(* IEC 61131-3 sources: SafePLC-Gen-Evaluation/Evaluation Results/P_ID/run_01, 2 files *)

(* ---- io_declarations.st ---- *)
(* ==================================================  *)
(* PLC I/O Variable Declarations — CODESYS 3.5  *)
(* Generated by SafePLC-Gen Multimodal  *)
(* ==================================================  *)

VAR_GLOBAL
    (* --- Analog Inputs ---  *)
    FT_10_Raw                    AT %IW0       : INT := 0;    (* FT-10 — Flow transmitter on upper feed line, mea  *)
    FT_11_Raw                    AT %IW2       : INT := 0;    (* FT-11 — Flow transmitter on lower feed line, mea  *)
    (* --- Analog Outputs ---  *)
    Fv_3_3040_Out                AT %QW0       : INT := 0;    (* Fv-3-3040 — Flow control valve on upper feed line fr  *)
    Fv_3_3041_Out                AT %QW2       : INT := 0;    (* Fv-3-3041 — Flow control valve on lower feed line fr  *)
END_VAR

(* ---- generated_code.st ---- *)
(* Generated by SafePLC-Gen Multimodal — CODESYS 3.5 *)
(* IEC 61131-3 Structured Text *)
(* Date: 2026-04-25T12:45:35.863016 *)

PROGRAM FlowControl

VAR
    FT_10_Raw                    AT %IW0       : INT := 0;
    FT_11_Raw                    AT %IW2       : INT := 0;
    Fv_3_3040_Out                AT %QW0       : INT := 0;
    Fv_3_3041_Out                AT %QW2       : INT := 0;
END_VAR

VAR
    FT_10_Scaled                 : REAL := 0.0;
    FT_11_Scaled                 : REAL := 0.0;

    FT_10_HH_SP                  : REAL := 180.0;
    FT_10_H_SP                   : REAL := 160.0;
    FT_10_L_SP                   : REAL := 40.0;
    FT_10_LL_SP                  : REAL := 20.0;
    FT_10_Deadband               : REAL := 5.0;
    FT_10_H                      : BOOL := FALSE;
    FT_10_L                      : BOOL := FALSE;
    FT_10_HH_Latch               : SR := (S1 := FALSE, R := FALSE, Q1 := FALSE);
    FT_10_LL_Latch               : SR := (S1 := FALSE, R := FALSE, Q1 := FALSE);
    FT_10_HH_Ack                 : BOOL := FALSE;
    FT_10_LL_Ack                 : BOOL := FALSE;

    FT_11_HH_SP                  : REAL := 180.0;
    FT_11_H_SP                   : REAL := 160.0;
    FT_11_L_SP                   : REAL := 40.0;
    FT_11_LL_SP                  : REAL := 20.0;
    FT_11_Deadband               : REAL := 5.0;
    FT_11_H                      : BOOL := FALSE;
    FT_11_L                      : BOOL := FALSE;
    FT_11_HH_Latch               : SR := (S1 := FALSE, R := FALSE, Q1 := FALSE);
    FT_11_LL_Latch               : SR := (S1 := FALSE, R := FALSE, Q1 := FALSE);
    FT_11_HH_Ack                 : BOOL := FALSE;
    FT_11_LL_Ack                 : BOOL := FALSE;

    FT_10_SP                     : REAL := 100.0;
    FT_10_Kp                     : REAL := 1.2;
    FT_10_Ki                     : REAL := 0.05;
    FT_10_Error                  : REAL := 0.0;
    FT_10_Integral               : REAL := 0.0;
    FT_10_Output                 : REAL := 0.0;

    FT_11_SP                     : REAL := 100.0;
    FT_11_Kp                     : REAL := 1.2;
    FT_11_Ki                     : REAL := 0.05;
    FT_11_Error                  : REAL := 0.0;
    FT_11_Integral               : REAL := 0.0;
    FT_11_Output                 : REAL := 0.0;

    System_Alarm                 : BOOL := FALSE;
    FirstScan                    : BOOL := TRUE;
END_VAR

IF FirstScan THEN
    Fv_3_3040_Out  := 6554;
    Fv_3_3041_Out  := 6554;
    FT_10_Integral := 0.0;
    FT_11_Integral := 0.0;
    FirstScan      := FALSE;
    RETURN;
END_IF;

FT_10_Scaled := ((INT_TO_REAL(FT_10_Raw) - 6554.0) / (32767.0 - 6554.0)) * 200.0;
FT_11_Scaled := ((INT_TO_REAL(FT_11_Raw) - 6554.0) / (32767.0 - 6554.0)) * 200.0;

(* FT-10 HH latch *)
IF FT_10_Scaled >= FT_10_HH_SP THEN
    FT_10_HH_Latch.S1 := TRUE;
ELSIF FT_10_Scaled <= (FT_10_HH_SP - FT_10_Deadband) THEN
    FT_10_HH_Latch.S1 := FALSE;
END_IF;
FT_10_HH_Latch.R := FT_10_HH_Ack AND (FT_10_Scaled < FT_10_HH_SP);
FT_10_HH_Latch(S1 := FT_10_HH_Latch.S1, R := FT_10_HH_Latch.R);

(* FT-10 H alarm *)
IF FT_10_Scaled >= FT_10_H_SP THEN
    FT_10_H := TRUE;
ELSIF FT_10_Scaled <= (FT_10_H_SP - FT_10_Deadband) THEN
    FT_10_H := FALSE;
END_IF;

(* FT-10 L alarm *)
IF FT_10_Scaled <= FT_10_L_SP THEN
    FT_10_L := TRUE;
ELSIF FT_10_Scaled >= (FT_10_L_SP + FT_10_Deadband) THEN
    FT_10_L := FALSE;
END_IF;

(* FT-10 LL latch *)
IF FT_10_Scaled <= FT_10_LL_SP THEN
    FT_10_LL_Latch.S1 := TRUE;
ELSIF FT_10_Scaled >= (FT_10_LL_SP + FT_10_Deadband) THEN
    FT_10_LL_Latch.S1 := FALSE;
END_IF;
FT_10_LL_Latch.R := FT_10_LL_Ack AND (FT_10_Scaled > FT_10_LL_SP);
FT_10_LL_Latch(S1 := FT_10_LL_Latch.S1, R := FT_10_LL_Latch.R);

(* FT-11 HH latch *)
IF FT_11_Scaled >= FT_11_HH_SP THEN
    FT_11_HH_Latch.S1 := TRUE;
ELSIF FT_11_Scaled <= (FT_11_HH_SP - FT_11_Deadband) THEN
    FT_11_HH_Latch.S1 := FALSE;
END_IF;
FT_11_HH_Latch.R := FT_11_HH_Ack AND (FT_11_Scaled < FT_11_HH_SP);
FT_11_HH_Latch(S1 := FT_11_HH_Latch.S1, R := FT_11_HH_Latch.R);

(* FT-11 H alarm *)
IF FT_11_Scaled >= FT_11_H_SP THEN
    FT_11_H := TRUE;
ELSIF FT_11_Scaled <= (FT_11_H_SP - FT_11_Deadband) THEN
    FT_11_H := FALSE;
END_IF;

(* FT-11 L alarm *)
IF FT_11_Scaled <= FT_11_L_SP THEN
    FT_11_L := TRUE;
ELSIF FT_11_Scaled >= (FT_11_L_SP + FT_11_Deadband) THEN
    FT_11_L := FALSE;
END_IF;

(* FT-11 LL latch *)
IF FT_11_Scaled <= FT_11_LL_SP THEN
    FT_11_LL_Latch.S1 := TRUE;
ELSIF FT_11_Scaled >= (FT_11_LL_SP + FT_11_Deadband) THEN
    FT_11_LL_Latch.S1 := FALSE;
END_IF;
FT_11_LL_Latch.R := FT_11_LL_Ack AND (FT_11_Scaled > FT_11_LL_SP);
FT_11_LL_Latch(S1 := FT_11_LL_Latch.S1, R := FT_11_LL_Latch.R);

(* PI control — upper loop *)
FT_10_Error    := FT_10_SP - FT_10_Scaled;
FT_10_Integral := FT_10_Integral + (FT_10_Ki * FT_10_Error);
IF FT_10_Integral > 100.0 THEN
    FT_10_Integral := 100.0;
ELSIF FT_10_Integral < 0.0 THEN
    FT_10_Integral := 0.0;
END_IF;
FT_10_Output := (FT_10_Kp * FT_10_Error) + FT_10_Integral;
IF FT_10_Output > 100.0 THEN
    FT_10_Output := 100.0;
ELSIF FT_10_Output < 0.0 THEN
    FT_10_Output := 0.0;
END_IF;
Fv_3_3040_Out := REAL_TO_INT(6554.0 + (FT_10_Output / 100.0) * (32767.0 - 6554.0));

(* PI control — lower loop *)
FT_11_Error    := FT_11_SP - FT_11_Scaled;
FT_11_Integral := FT_11_Integral + (FT_11_Ki * FT_11_Error);
IF FT_11_Integral > 100.0 THEN
    FT_11_Integral := 100.0;
ELSIF FT_11_Integral < 0.0 THEN
    FT_11_Integral := 0.0;
END_IF;
FT_11_Output := (FT_11_Kp * FT_11_Error) + FT_11_Integral;
IF FT_11_Output > 100.0 THEN
    FT_11_Output := 100.0;
ELSIF FT_11_Output < 0.0 THEN
    FT_11_Output := 0.0;
END_IF;
Fv_3_3041_Out := REAL_TO_INT(6554.0 + (FT_11_Output / 100.0) * (32767.0 - 6554.0));

System_Alarm :=
    FT_10_HH_Latch.Q1 OR FT_10_LL_Latch.Q1 OR FT_10_H OR FT_10_L OR
    FT_11_HH_Latch.Q1 OR FT_11_LL_Latch.Q1 OR FT_11_H OR FT_11_L;

END_PROGRAM
